FUNCTION_BLOCK FB_RS_COMM_NO_SIM EXTENDS FB_RS_COMM_BASE
VAR_INPUT
END_VAR
VAR_OUTPUT
END_VAR
VAR CONSTANT
END_VAR
VAR
	{attribute 'OPC.UA.DA' := '1'}
	cfg:		T_RS_COMM_CFG;				// Config parameters
	{attribute 'OPC.UA.DA' := '1'}
	ctrl:		T_RS_COMM_CTRL;				// Control parameters
	{attribute 'OPC.UA.DA' := '1'}
	{attribute 'OPC.UA.DA.Access' := '1'}
	info:		T_RS_COMM_INFO; 			// Info parameters - ReadOnly
	{attribute 'OPC.UA.DA' := '1'}
	{attribute 'OPC.UA.DA.Access' := '1'}
	stat:		T_RS_COMM_STAT;				// Status parameters - ReadOnly

	sim:		FB_SIM_RS_COMM_BASE;		// COMM simulator

	// Physical signals - to be mapped to EL60xx serial port controller !!!
	COMin_EL60xx	AT %I* 	: KL6inData22B;	(* linked to the EL60xx *)
	COMout_EL60xx	AT %Q*	: KL6outData22B;(* linked to the EL60xx *)

	(* Serial line control *)
	COMportControl: 		SerialLineControl;

END_VAR

// Set references
cfgRef	REF=cfg;
ctrlRef	REF=ctrl;
infoRef	REF=info;
statRef	REF=stat;
simRef	REF=sim;

SUPER^();

METHOD M_ActionInitExecute
VAR_INPUT
END_VAR
//
// Copy input parameters to cfg
//
cfg.sCmdSuffix		:= in_sCmdSuffix;
cfg.sReplySuffix	:= in_sReplySuffix;
cfg.nTimeout		:= in_nTimeout;

//
// If in simulation, there is no need to reset anything.
// Just set it to initialised and go to IDLE state.
//
IF in_bSimulation THEN
	fbTimer (IN := FALSE);
	statRef.bInitialised	:= TRUE;
	statRef.nStatus			:= E_RS_COMM_STATUS.IDLE;
	statRef.sStatus			:= 'INITIALISED';
	State 					:= E_RS_COMM_STATE.IDLE;
ELSE
	stat.bInitialised	:= FALSE;
	stat.sStatus		:= 'INITIALISING';
	stat.nStatus		:= E_RS_COMM_STATUS.BUSY;
	stat.sReply 		:= ''; (* No reply yet *)
	stat.nErrorCode		:= E_RS_COMM_ERROR.OK;
	stat.sErrorText		:= 'OK';
	
	// Reset the connected serial hardware 
	ComReset (
		Execute 	:= FALSE,
		pComIn		:= ADR(COMin_EL60xx),
		pComOut		:= ADR(COMout_EL60xx),
		SizeComIn	:= SIZEOF(COMin_EL60xx),
		);
	
	// Set next state
	State 	:= E_RS_COMM_STATE.RESET;
END_IF
END_METHOD

METHOD M_ComPortControl
VAR_INPUT
END_VAR
// RS specific call of the background communication process
COMportControl(
	Mode		:= ComSerialLineMode_t.SERIALLINEMODE_KL6_22B_STANDARD,
	pComIn		:= ADR(COMin_EL60xx),					(* I/O data; see global variables *)
	pComOut		:= ADR(COMout_EL60xx),					(* I/O data; see global variables *)
	SizeComIn	:= UINT_TO_INT(SIZEOF(COMin_EL60xx)),	(* I/O data; see global variables *)
	TxBuffer	:= TxBuffer,							(* transmit buffer; see global variables *)
	RxBuffer	:= RxBuffer);							(* receive buffer; see global variables *)
END_METHOD

METHOD M_Reset
VAR_INPUT
END_VAR
// RS specific call of communication reset
//
// Reset the connected serial hardware.
ComReset (
	Execute 	:= TRUE,
	pComIn		:= ADR(COMin_EL60xx),
	pComOut		:= ADR(COMout_EL60xx),
	SizeComIn	:= SIZEOF(COMin_EL60xx),
	);

(* Next step is to clear the buffers *)
IF ComReset.Done THEN
	fbTimer (IN := FALSE);	// Reset the timer
	State 		:= E_RS_COMM_STATE.CLEAR_BUFFER;
END_IF
END_METHOD

END_FUNCTION_BLOCK

(* stored: Version 1.1.0.1, ProductVersion 3.1.4024.3
   POU FB_RS_COMM_NO_SIM: Id {3fa7d2d2-bfdb-4d28-bdd3-2e164c05ef18}, SpecialFunc None
   Method M_ActionInitExecute: Id {3ae426a9-72cc-48ad-a9ff-dd538ce057e2}
   Method M_ComPortControl: Id {fc4137c2-f814-4172-9a96-94fa39a82306}
   Method M_Reset: Id {4534819d-7a5e-461f-938b-c29dc65b00c3} *)
